FUNCTION_BLOCK FB_VISU_CYLINDER
VAR_INPUT
END_VAR
VAR_OUTPUT
END_VAR
VAR
	itfPneuActor: I_PNEU_ACTOR;	
	itfOpMode: I_OP_MODE;
	iMove: INT;
	iNegMove: INT;
	iMoveSmall: INT;
	iNegMoveSmall: INT;
	iAngle: INT;
	iNegAngle: INT;
	strInfo: STRING;
	strFullObjName: STRING;
	bMoveToBase: BOOL;
	bMoveToWork: BOOL;
	bAllOff: BOOL;
	bInBasePos: BOOL;
	bInWorkPos: BOOL;
	bInMidPos: 	BOOL;
	bFaultWorkPos: BOOL;
	bFaultBasePos: BOOL;
	dwFrameColorBase: DWORD:= 16#FF00BFFF;
	dwFrameColorWork: DWORD:= 16#FF00BFFF;
	dwFrameColorMid: DWORD:= 16#FF00BFFF;
	bBaseArrowInvisible: BOOL:=TRUE;
	bWorkArrowInvisible: BOOL:=TRUE;
	bMidkArrowInvisible: BOOL:=TRUE;
	iFrame: INT;
	bFrameInvisible: BOOL:= TRUE;
	stEvent: ST_EVENT;
	dwColor: DWORD;
END_VAR

IF NOT (itfOpMode.P_OP_MODE_STATE=OP_MODE.MANUAL) THEN
	bFrameInvisible:= TRUE;
END_IF

IF (itfPneuActor.P_State=E_POS_STATE.MoveToBase) THEN
//IF bMoveToBase AND NOT bInBasePos THEN
	iMove:=-30;
	iAngle:=-90;
	//strInfo:= 'Zylinder fährt in Grundposition';
	strInfo:= F_RET_TXTLIST_ENTRY(strPortNr:= '851', strID:='3', strTxtLstName:= 'TXT_LIST_PNEMATIC_ACTOR');
	//bMoveToWork:= FALSE;
	dwFrameColorBase:= 16#FFFFA500;
	bBaseArrowInvisible:= FALSE;
	bWorkArrowInvisible:=TRUE;	
	bMidkArrowInvisible:=TRUE;
END_IF

IF (itfPneuActor.P_State=E_POS_STATE.InBasePos) THEN
//IF bMoveToBase AND bInBasePos THEN
	iMove:=0;
	iAngle:=0;
	//strInfo:= 'Zylinder ist in Grundposition';
	strInfo:= F_RET_TXTLIST_ENTRY(strPortNr:= '851', strID:='4', strTxtLstName:= 'TXT_LIST_PNEMATIC_ACTOR');
	//bMoveToWork:= FALSE;
	dwFrameColorBase:= 16#FF77BB77;
	bBaseArrowInvisible:= FALSE;
	bWorkArrowInvisible:=TRUE;	
	bMidkArrowInvisible:=TRUE;
END_IF

IF (itfPneuActor.P_State=E_POS_STATE.MoveToWork) THEN
//IF bMoveToWork AND NOT bInworkPos THEN
	iMove:=-30;
	iAngle:=-90;
	//strInfo:= 'Zylinder fährt in Arbeitsposition';
	strInfo:= F_RET_TXTLIST_ENTRY(strPortNr:= '851', strID:='5', strTxtLstName:= 'TXT_LIST_PNEMATIC_ACTOR');
	//bMoveToBase:= FALSE;
	dwFrameColorwork:= 16#FFFFA500;
	bBaseArrowInvisible:= TRUE;
	bWorkArrowInvisible:=FALSE;	
	bMidkArrowInvisible:=TRUE;
END_IF

IF (itfPneuActor.P_State=E_POS_STATE.InWorkPos) THEN
//IF bMoveToWork AND bInWorkPos THEN
	iMove:=-70;
	iAngle:=180;
	//strInfo:= 'Zylinder ist in Arbeitsposition';
	strInfo:= F_RET_TXTLIST_ENTRY(strPortNr:= '851', strID:='6', strTxtLstName:= 'TXT_LIST_PNEMATIC_ACTOR');
	//bMoveTobase:= FALSE;
	dwFrameColorWork:= 16#FF77BB77;
	bBaseArrowInvisible:= TRUE;
	bWorkArrowInvisible:=FALSE;	
	bMidkArrowInvisible:=TRUE;
END_IF

IF (itfPneuActor.P_State=E_POS_STATE.InMidPos) THEN
//IF bMoveToWork AND bInWorkPos THEN
	iMove:=-50;
	iAngle:=-90;
	//strInfo:= 'Zylinder ist in Arbeitsposition';
	strInfo:= F_RET_TXTLIST_ENTRY(strPortNr:= '851', strID:='15', strTxtLstName:= 'TXT_LIST_PNEMATIC_ACTOR');
	//bMoveTobase:= FALSE;
	dwFrameColorMid:= 16#FF77BB77;
	bBaseArrowInvisible:= TRUE;
	bWorkArrowInvisible:=TRUE;	
	bMidkArrowInvisible:=FALSE;
END_IF

IF (itfPneuActor.P_State=E_POS_STATE.NoDefPos) THEN
//IF bMoveToWork AND bInWorkPos THEN
	iMove:=-30;
	iNegAngle:=-90;
	//strInfo:= 'Zylinder in undefinierter Position';
	strInfo:= F_RET_TXTLIST_ENTRY(strPortNr:= '851', strID:='7', strTxtLstName:= 'TXT_LIST_PNEMATIC_ACTOR');
	//bMoveTobase:= FALSE;
	dwFrameColorWork:= 16#FF77BB77;
	bBaseArrowInvisible:= TRUE;
	bWorkArrowInvisible:=TRUE;	
	bMidkArrowInvisible:=TRUE;
END_IF

IF (itfPneuActor.P_State=E_POS_STATE.TimeOutToBase) THEN
//IF bMoveToWork AND bInWorkPos THEN
	iMove:=-30;
	iAngle:=-90;
	//strInfo:= 'Timeout bei Fahrt nach Grundstellung';
	strInfo:= F_RET_TXTLIST_ENTRY(strPortNr:= '851', strID:='8', strTxtLstName:= 'TXT_LIST_PNEUMATIC_ACTOR');
	//bMoveTobase:= FALSE;
	dwFrameColorWork:= 16#FFFF00FF;
	bBaseArrowInvisible:= TRUE;
	bWorkArrowInvisible:=FALSE;	
	bMidkArrowInvisible:=TRUE;
END_IF

IF (itfPneuActor.P_State=E_POS_STATE.TimeOutToWork) THEN
//IF bMoveToWork AND bInWorkPos THEN
	iMove:=-30;	
	iAngle:=-90;
	//strInfo:= 'Timeout bei Fahrt nach Arbeitsstellung';
	strInfo:= F_RET_TXTLIST_ENTRY(strPortNr:= '851', strID:='9', strTxtLstName:= 'TXT_LIST_PNEUMATIC_ACTOR');
	//bMoveTobase:= FALSE;
	dwFrameColorWork:= 16#FFFF00FF;
	bBaseArrowInvisible:= FALSE;
	bWorkArrowInvisible:=TRUE;	
	bMidkArrowInvisible:=TRUE;
END_IF

IF  (itfPneuActor.P_State=E_POS_STATE.MoveToWorkLock) THEN
	strInfo:= stEvent.strEventText;
	dwFrameColorWork:= Color.dwRed;
	bBaseArrowInvisible:= TRUE;
	bWorkArrowInvisible:=FALSE;	
	bMidkArrowInvisible:=TRUE;
END_IF

IF (itfPneuActor.P_State=E_POS_STATE.MoveToBaseLock) THEN
	strInfo:= stEvent.strEventText;
	dwFrameColorBase:= Color.dwRed;
	bBaseArrowInvisible:= FALSE;
	bWorkArrowInvisible:=TRUE;	
	bMidkArrowInvisible:=TRUE;
END_IF

strFullObjName:= itfPneuActor.P_FullObjectPath;

IF (itfOpMode.P_OP_MODE_STATE=OP_MODE.MANUAL) THEN
	IF bMoveToBase THEN
		itfPneuActor.M_ToBasePos();
		bMoveToBase:=FALSE;
		//bMoveToWork:= FALSE;
		//bAllOff:= FALSE;
	END_IF
	IF bMoveToWork THEN
		itfPneuActor.M_ToWorkPos();
		//bMoveToBase:=FALSE;
		bMoveToWork:= FALSE;
		//bAllOff:= FALSE;
	END_IF
	IF bAllOff THEN
		itfPneuActor.M_Stop();
		//bMoveToBase:=FALSE;
		//bMoveToWork:= FALSE;
		bAllOff:= FALSE;
	END_IF
	
ELSE
	bMoveToBase:=FALSE;
	bMoveToWork:= FALSE;
    bAllOff:= FALSE;
END_IF



iNegMove:= iMove*(-1);
iNegAngle:=iAngle*(-1);
iMoveSmall:=iMove/2;
iNegMoveSmall:=iNegMove/2;
stEvent:= itfPneuActor.P_Event;

IF stEvent.bEventActive THEN
	dwColor:= Color.dwOrange;
END_IF

METHOD FB_init : BOOL
VAR_INPUT
	bInitRetains : BOOL; // if TRUE, the retain variables are initialized (warm start / cold start)
	bInCopyCode : BOOL;  // if TRUE, the instance afterwards gets moved into the copy code (online change)
	itfPneuActor: I_PNEU_ACTOR;
	itfOpMode: I_OP_MODE;
END_VAR
THIS^.itfPneuActor:= itfPneuActor;
THIS^.itfOpMode:= itfOpMode;
END_METHOD

END_FUNCTION_BLOCK

(* stored: Version 1.1.0.1, ProductVersion 3.1.4024.12
   POU FB_VISU_CYLINDER: Id {bda66ac4-9025-485b-94cc-b133d7ffc625}, SpecialFunc None
   Method FB_init: Id {fe04a5a7-319d-43de-bad4-3c0095cd9fbe} *)
